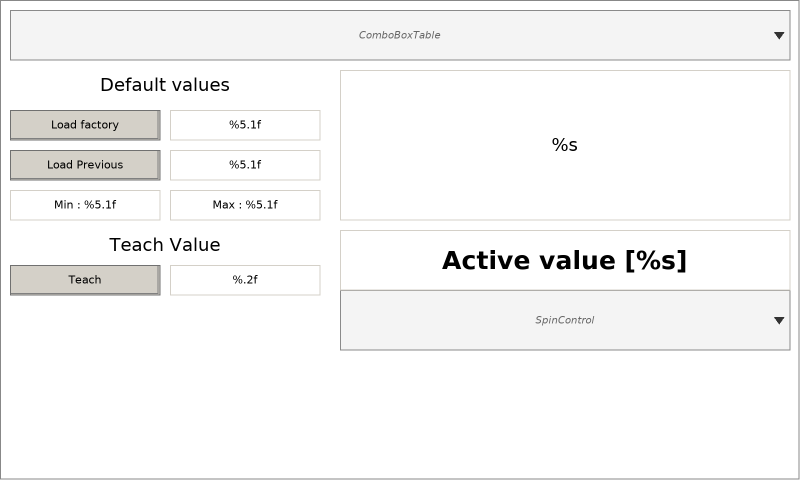
VISUALIZATION ParameterControl  // 800x480
    ComboBoxTable (10,10 780x50), variable: GVL_Parameters.fbParameterHandler.nLookupIndex, data array: GVL_Parameters.fbParameterHandler.arParameters
        p1128707560: GVL_Parameters.fbParameterHandler.nNumberOfParameters
        p3854506369: GVL_Parameters.fbParameterHandler.arParameters[INDEX].nNumber
        p1892666644: GVL_Parameters.fbParameterHandler.arParameters[INDEX].sName
        p338671338: GVL_Parameters.fbParameterHandler.arParameters[INDEX].sType
        p2170511999: GVL_Parameters.fbParameterHandler.arParameters[INDEX].pParameter^
    Group (10,70 310x150)
        Button (0,40 150x30), "Load factory"
            tap GVL_Parameters.fbParameterHandler.bCmdLoadfactory
        Label (0,0 310x30), "Default values"
        Textfield (160,40 150x30), "%5.1f", text variable: GVL_Parameters.fbParameterHandler.arParameters[GVL_Parameters.fbParameterHandler.nLookupIndex].pParameter^.fFactory
            OnMouseClick: write the text variable via VisuDialogs.Numpad, min GVL_Parameters.fbParameterHandler.arParameters[GVL_Parameters.fbParameterHandler.nLookupIndex].pParameter^.fMinimum, max GVL_Parameters.fbParameterHandler.arParameters[GVL_Parameters.fbParameterHandler.nLookupIndex].pParameter^.fMaximum
        Button (0,80 150x30), "Load Previous"
            tap GVL_Parameters.fbParameterHandler.bCmdLoadFromPrevious
        Textfield (160,80 150x30), "%5.1f", text variable: GVL_Parameters.fbParameterHandler.arParameters[GVL_Parameters.fbParameterHandler.nLookupIndex].pParameter^.fSaved
        Textfield (160,120 150x30), "Max : %5.1f", text variable: GVL_Parameters.fbParameterHandler.arParameters[GVL_Parameters.fbParameterHandler.nLookupIndex].pParameter^.fMaximum
            OnMouseClick: write the text variable via VisuDialogs.Numpad
        Textfield (0,120 150x30), "Min : %5.1f", text variable: GVL_Parameters.fbParameterHandler.arParameters[GVL_Parameters.fbParameterHandler.nLookupIndex].pParameter^.fMinimum
            OnMouseClick: write the text variable via VisuDialogs.Numpad
    Textfield (340,70 450x150), "%s", text variable: GVL_Parameters.fbParameterHandler.arParameters[GVL_Parameters.fbParameterHandler.nLookupIndex].pParameter^.sDiscription
    SpinControl (340,290 450x60), variable: GVL_Parameters.fbParameterHandler.arParameters[GVL_Parameters.fbParameterHandler.nLookupIndex].pParameter^.fValue
        p576042468: GVL_Parameters.fbParameterHandler.arParameters[GVL_Parameters.fbParameterHandler.nLookupIndex].pParameter^.fMinimum
        p651134158: GVL_Parameters.fbParameterHandler.arParameters[GVL_Parameters.fbParameterHandler.nLookupIndex].pParameter^.fMaximum
        OnMouseClick: write the text variable via VisuDialogs.Numpad, min GVL_Parameters.fbParameterHandler.arParameters[GVL_Parameters.fbParameterHandler.nLookupIndex].pParameter^.fMinimum, max GVL_Parameters.fbParameterHandler.arParameters[GVL_Parameters.fbParameterHandler.nLookupIndex].pParameter^.fMaximum
    Textfield (340,230 450x60), "Active value [%s]", text variable: GVL_Parameters.fbParameterHandler.arParameters[GVL_Parameters.fbParameterHandler.nLookupIndex].pParameter^.sUnit
    Group (10,230 310x65)
        Label (0,0 310x30), "Teach Value"
        Textfield (160,35 150x30), "%.2f", text variable: GVL_Parameters.fbParameterHandler.arParameters[GVL_Parameters.fbParameterHandler.nLookupIndex].pParameter^.fPrepared
        Button (0,35 150x30), "Teach"
            tap GVL_Parameters.fbParameterHandler.bCmdAcceptTeach
END_VISUALIZATION

(* stored: Version 1.1.0.1, ProductVersion 3.1.4024.9
   Visu ParameterControl: Id {19588bb2-b793-42b3-8298-3e4d21977e8c} *)
